SUBAPPLICATION Uebung_076_AUI (* MSS mit Compound Scaling auf UT ausgeben (Adapter Version) *)
  (* Standard: 61499-2; Description: Copyright (c) 2023 Meisterschulen am Ostbahnhof This program and the accompanying materials are made available under the terms of the Eclipse Public License 2.0 which is available at https://www.eclipse.org/legal/epl-2.0/ SPDX-License-Identifier: EPL-2.0 *)
  (* Version 1.1, 2026-09-17, Franz Höpfinger, Meisterschulen am Ostbahnhof, Diese sub hat einen Bug. für einen Fix: siehe Uebung_076a_AUI.SUB *)
  (* Version 1.0, 2026-06-01, Franz Höpfinger, Meisterschulen am Ostbahnhof, MSS Machine Selected Speed mit Compound Scaling (Adapter Version) *)
  PACKAGE Uebungen;
  IMPORT Uebungen::const::UT::TECU::DefaultPool_TECU_Numeric::NumberVariable_Wheel_based_machine_speed_N;
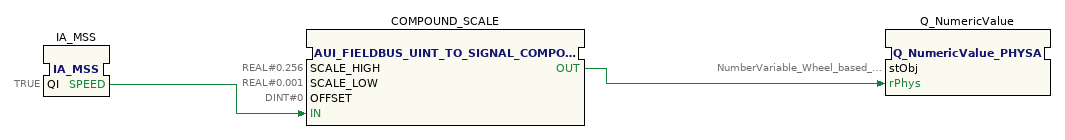
  (* TODO: NumberVariable_Machine_selected_speed im Object Pool anlegen, und hier umändern. solange verwenden wir hier NumberVariable_Wheel_based_machine_speed ersatzweise *)
  FBS
    IA_MSS : isobus::tecu::IA_MSS(QI := TRUE);
    COMPOUND_SCALE : logiBUS::signalprocessing::fieldbus::AUI_FIELDBUS_UINT_TO_SIGNAL_COMPOUND_SCALE(SCALE_HIGH := REAL#0.256, SCALE_LOW := REAL#0.001, OFFSET := DINT#0);
    Q_NumericValue : isobus::UT::Q::Q_NumericValue_PHYSA(stObj := NumberVariable_Wheel_based_machine_speed_N);
  END_FBS
  ADAPTER_CONNECTIONS
    IA_MSS.SPEED TO COMPOUND_SCALE.IN;
    COMPOUND_SCALE.OUT TO Q_NumericValue.rPhys;
  END_CONNECTIONS
END_SUBAPPLICATION
